// TwinCAT 3 PLC project Gantry
// ProgramVersion: 3.1.4023.0
// libraries:
//   Tc2_MC2, * (Beckhoff Automation GmbH)
//   Tc2_Standard, * (Beckhoff Automation GmbH)
//   Tc2_System, * (Beckhoff Automation GmbH)
//   Tc3_Module, * (Beckhoff Automation GmbH)
// project tree:
//   DUTs/ ST_PalletRecord.TcDUT
//   GVLs/ GVL_IO.TcGVL
//   / PlcTask.TcTTO
//   POUs/Devices/Actuator/ E_ActuatorCommand.TcDUT, E_ActuatorState.TcDUT, FB_Actuator.TcPOU
//   POUs/Devices/Axis/ E_AxisCommand.TcDUT, E_AxisState.TcDUT, FB_Axis.TcPOU
//   POUs/Devices/RFID/ E_RFIDCommand.TcDUT, E_RFIDState.TcDUT, FB_RFID.TcPOU
//   POUs/Interfaces/ I_GantryPallet.TcIO, I_GantryPart.TcIO
//   POUs/Modules/Gantry/ E_GantryCommand.TcDUT, E_GantryState.TcDUT, FB_Gantry.TcPOU
//   POUs/Modules/PalletStation/ E_PalletStationCommand.TcDUT, E_PalletStationState.TcDUT, FB_PalletStation.TcPOU
//   POUs/Modules/PartStation/ E_PartStationCommand.TcDUT, E_PartStationState.TcDUT, FB_PartStation.TcPOU
//   Program/ MAIN.TcPOU
// real-time tasks:
//   TASK PlcTask: cycle T#10ms, priority 20, ADS port 350
// motion (NC):
//   TASK NC-Task 1 SAF: cycle T#2ms, priority 4, ADS port 501
//   TASK NC-Task 1 SVB: cycle T#10ms, priority 8, ADS port 511
//   AXIS Gantry1X (id 1)
//     OtherSettings: AllowMotionCmdToSlave=true
//     encoder EncType=1
//     drive DrvType=5
//       Analog: TorqueSetpointScale=10, ScaleFactorActTorque=0.1
//       TimeComp: TaskDelayCycles=1
//     controller CtrType=1
//       CtrPara: PriorControlFactor=1
//         Observer: BandWidth=20
//   AXIS Gantry1Z (id 2)
//     OtherSettings: AllowMotionCmdToSlave=true
//     encoder EncType=1
//     drive DrvType=5
//       Analog: TorqueSetpointScale=10, ScaleFactorActTorque=0.1
//       TimeComp: TaskDelayCycles=1
//     controller CtrType=1
//       CtrPara: PriorControlFactor=1
//         Observer: BandWidth=20
//   AXIS Gantry2X (id 3)
//     OtherSettings: AllowMotionCmdToSlave=true
//     encoder EncType=1
//     drive DrvType=5
//       Analog: TorqueSetpointScale=10, ScaleFactorActTorque=0.1
//       TimeComp: TaskDelayCycles=1
//     controller CtrType=1
//       CtrPara: PriorControlFactor=1
//         Observer: BandWidth=20
//   AXIS Gantry2Z (id 4)
//     OtherSettings: AllowMotionCmdToSlave=true
//     encoder EncType=1
//     drive DrvType=5
//       Analog: TorqueSetpointScale=10, ScaleFactorActTorque=0.1
//       TimeComp: TaskDelayCycles=1
//     controller CtrType=1
//       CtrPara: PriorControlFactor=1
//         Observer: BandWidth=20
//   AXIS PalletConveyor (id 5)
//     OtherSettings: AllowMotionCmdToSlave=true
//     encoder EncType=1
//     drive DrvType=5
//       Analog: TorqueSetpointScale=10, ScaleFactorActTorque=0.1
//       TimeComp: TaskDelayCycles=1
//     controller CtrType=1
//       CtrPara: PriorControlFactor=1
//         Observer: BandWidth=20
//   AXIS PartConveyor1 (id 6)
//     OtherSettings: AllowMotionCmdToSlave=true
//     encoder EncType=1
//     drive DrvType=5
//       Analog: TorqueSetpointScale=10, ScaleFactorActTorque=0.1
//       TimeComp: TaskDelayCycles=1
//     controller CtrType=1
//       CtrPara: PriorControlFactor=1
//         Observer: BandWidth=20
//   AXIS PartConveyor2 (id 7)
//     OtherSettings: AllowMotionCmdToSlave=true
//     encoder EncType=1
//     drive DrvType=5
//       Analog: TorqueSetpointScale=10, ScaleFactorActTorque=0.1
//       TimeComp: TaskDelayCycles=1
//     controller CtrType=1
//       CtrPara: PriorControlFactor=1
//         Observer: BandWidth=20
// variable links:
//   Gantry/Gantry Instance <-> NC-Task 1 SAF/Axes/Gantry1X
//     PlcTask Inputs/GVL_IO.Gantry1X.NcToPlc <-> Outputs/ToPlc
//     PlcTask Outputs/GVL_IO.Gantry1X.PlcToNc <-> Inputs/FromPlc
//   Gantry/Gantry Instance <-> NC-Task 1 SAF/Axes/Gantry1Z
//     PlcTask Inputs/GVL_IO.Gantry1Z.NcToPlc <-> Outputs/ToPlc
//     PlcTask Outputs/GVL_IO.Gantry1Z.PlcToNc <-> Inputs/FromPlc
//   Gantry/Gantry Instance <-> NC-Task 1 SAF/Axes/Gantry2X
//     PlcTask Inputs/GVL_IO.Gantry2X.NcToPlc <-> Outputs/ToPlc
//     PlcTask Outputs/GVL_IO.Gantry2X.PlcToNc <-> Inputs/FromPlc
//   Gantry/Gantry Instance <-> NC-Task 1 SAF/Axes/Gantry2Z
//     PlcTask Inputs/GVL_IO.Gantry2Z.NcToPlc <-> Outputs/ToPlc
//     PlcTask Outputs/GVL_IO.Gantry2Z.PlcToNc <-> Inputs/FromPlc
//   Gantry/Gantry Instance <-> NC-Task 1 SAF/Axes/PalletConveyor
//     PlcTask Inputs/GVL_IO.PalletConveyor.NcToPlc <-> Outputs/ToPlc
//     PlcTask Outputs/GVL_IO.PalletConveyor.PlcToNc <-> Inputs/FromPlc
//   Gantry/Gantry Instance <-> NC-Task 1 SAF/Axes/PartConveyor1
//     PlcTask Inputs/GVL_IO.PartConveyor1.NcToPlc <-> Outputs/ToPlc
//     PlcTask Outputs/GVL_IO.PartConveyor1.PlcToNc <-> Inputs/FromPlc
//   Gantry/Gantry Instance <-> NC-Task 1 SAF/Axes/PartConveyor2
//     PlcTask Inputs/GVL_IO.PartConveyor2.NcToPlc <-> Outputs/ToPlc
//     PlcTask Outputs/GVL_IO.PartConveyor2.PlcToNc <-> Inputs/FromPlc

CONFIGURATION Gantry
    RESOURCE PLC ON TwinCAT3
        TASK PlcTask(INTERVAL := T#10ms, PRIORITY := 20);
        PROGRAM MAIN WITH PlcTask : MAIN;
    END_RESOURCE
END_CONFIGURATION

// ---- DUTs/ST_PalletRecord.TcDUT
TYPE ST_PalletRecord :
STRUCT
	ID				: STRING;
	Data			: ARRAY[1..100] OF STRING;
END_STRUCT
END_TYPE

// ---- POUs/Devices/Actuator/E_ActuatorCommand.TcDUT
{attribute 'qualified_only'}
{attribute 'strict'}
TYPE E_ActuatorCommand :
(
	None 		:= 0,
	Home		:= 1,
	Work		:= 2
) DINT;
END_TYPE

// ---- POUs/Devices/Actuator/E_ActuatorState.TcDUT
{attribute 'qualified_only'}
{attribute 'strict'}
TYPE E_ActuatorState :
(
	AtHome		:= 0, //Actuator at home
	AtWork		:= 1, //Actuator at work
	GoingToHome	:= 2, //Actuator going to home
	GoingToWork	:= 3 //Actuator going to work
) DINT;
END_TYPE

// ---- POUs/Devices/Axis/E_AxisCommand.TcDUT
{attribute 'qualified_only'}
{attribute 'strict'}
TYPE E_AxisCommand :
(
	None 				:= 0,
	TurnOn				:= 1,
	TurnOff				:= 2,
	ExecuteMoveAbs		:= 3,
	ExecuteMoveVel		:= 4,
	Stop				:= 5
) DINT;
END_TYPE

// ---- POUs/Devices/Axis/E_AxisState.TcDUT
{attribute 'qualified_only'}
{attribute 'strict'}
TYPE E_AxisState :
(
	Off					:= 0, //Axis is off
	Ready				:= 1, //Axis is ready/on
	Moving				:= 2, //Axis is moving to commanded position
	Stopping			:= 3, //Axis is stopping
	Stopped				:= 4, //Axis is stopped
	TurningOn			:= 5, //Axis is turning on
	TurningOff			:= 6 //Axis is turning off
) DINT;
END_TYPE

// ---- POUs/Devices/RFID/E_RFIDCommand.TcDUT
{attribute 'qualified_only'}
{attribute 'strict'}
TYPE E_RFIDCommand :
(
	None 		:= 0,
	Clear		:= 1,
	Read		:= 2
) DINT;
END_TYPE

// ---- POUs/Devices/RFID/E_RFIDState.TcDUT
{attribute 'qualified_only'}
{attribute 'strict'}
TYPE E_RFIDState :
(
	Idle			:= 0,
	Clearing		:= 1,
	Reading			:= 2,
	Completing		:= 3
);
END_TYPE

// ---- POUs/Modules/Gantry/E_GantryCommand.TcDUT
{attribute 'qualified_only'}
{attribute 'strict'}
TYPE E_GantryCommand :
(
	None 			:= 0,
	TurnOn			:= 1,
	TurnOff			:= 2,
	Pick			:= 3,
	Place			:= 4,
	Home			:= 5,
	Abort			:= 6
) DINT;
END_TYPE

// ---- POUs/Modules/Gantry/E_GantryState.TcDUT
{attribute 'qualified_only'}
{attribute 'strict'}
TYPE E_GantryState :
(
	Idle 			:= 0,
	TurningOn		:= 1,
	TurningOff		:= 2,
	Ready			:= 3,
	Picking			:= 4,
	Placing			:= 5,
	Homing			:= 6,
	Aborting		:= 7
) DINT;
END_TYPE

// ---- POUs/Modules/PalletStation/E_PalletStationCommand.TcDUT
{attribute 'qualified_only'}
{attribute 'strict'}
TYPE E_PalletStationCommand :
(
	None 			:= 0,
	Start			:= 1,
	Stop			:= 2,
	Home			:= 3,
	Abort			:= 4
) DINT;
END_TYPE

// ---- POUs/Modules/PalletStation/E_PalletStationState.TcDUT
{attribute 'qualified_only'}
{attribute 'strict'}
TYPE E_PalletStationState :
(
	Idle 			:= 0,
	Starting		:= 1,
	Running			:= 2,
	Stopping		:= 3,
	Homing			:= 4,
	Aborting		:= 5
);
END_TYPE

// ---- POUs/Modules/PartStation/E_PartStationCommand.TcDUT
{attribute 'qualified_only'}
{attribute 'strict'}
TYPE E_PartStationCommand :
(
	None 			:= 0,
	Start			:= 1,
	Stop			:= 2,
	Abort			:= 3
) DINT;
END_TYPE

// ---- POUs/Modules/PartStation/E_PartStationState.TcDUT
{attribute 'qualified_only'}
{attribute 'strict'}
TYPE E_PartStationState :
(
	Idle 			:= 0,
	Starting		:= 1,
	Running			:= 2,
	Stopping		:= 3,
	Stopped			:= 4,
	Aborting		:= 5
);
END_TYPE

// ---- GVLs/GVL_IO.TcGVL
{attribute 'qualified_only'}
VAR_GLOBAL
	Gantry1X			: AXIS_REF;
	Gantry1Z			: AXIS_REF;
	Gantry2X			: AXIS_REF;
	Gantry2Z			: AXIS_REF;
	PalletConveyor		: AXIS_REF;
	PartConveyor1		: AXIS_REF;
	PartConveyor2		: AXIS_REF;
	
	PalletRecord		: ARRAY[0..100] OF ST_PalletRecord;
	ActiveRecord		: DINT;
END_VAR

// ---- POUs/Interfaces/I_GantryPallet.TcIO
INTERFACE I_GantryPallet

PROPERTY PalletReady : BOOL
GET
END_GET
END_PROPERTY

END_INTERFACE

// ---- POUs/Interfaces/I_GantryPart.TcIO
INTERFACE I_GantryPart

PROPERTY PartPicked : BOOL
GET
END_GET
END_PROPERTY

PROPERTY PartReady : BOOL
GET
END_GET
END_PROPERTY

END_INTERFACE

// ---- Program/MAIN.TcPOU
PROGRAM MAIN
VAR
	inpSim					: BOOL := TRUE;
	
	PalletStation			: FB_PalletStation;
	Part1Station			: FB_PartStation;
	Part2Station			: FB_PartStation;
	Gantry1					: FB_Gantry;
	Gantry2					: FB_Gantry;
	
	Gantry1NextPlace		: DINT;
	Gantry2NextPlace		: DINT;
	
	Start					: BOOL;
	Abort					: BOOL;
	Home					: BOOL;
END_VAR

IF inpSim THEN
	Simulate();
END_IF

PalletStation(Axis := GVL_IO.PalletConveyor, 
		inpPalletRecord := GVL_IO.PalletRecord,
		inpActiveRecord := GVL_IO.ActiveRecord,
		ipGantry1 := Gantry1, 
		ipGantry2 := Gantry2);
Part1Station(Axis := GVL_IO.PartConveyor1, 
		ipGantry := Gantry1);
Part2Station(Axis := GVL_IO.PartConveyor2, 
		ipGantry := Gantry2);

Gantry1(AxisX := GVL_IO.Gantry1X,
		AxisZ := GVL_IO.Gantry1Z,
		ipPart := Part1Station,
		ipPallet := PalletStation,
		inpPalletRecord := GVL_IO.PalletRecord,
		inpActiveRecord := GVL_IO.ActiveRecord,
		inpDataIndex1 := 1,
		inpDataIndex2 := 2,
		inpDataIndex3 := 3,
		inpDataIndex4 := 4,
		inpDataIndex5 := 5,
		inpDataIndex6 := 6,
		inpX_HomePos := 0,		
		inpX_PickPos := 100,	
		inpX_PlacePos1 := 2050,
		inpX_PlacePos2 := 2100,
		inpX_PlacePos3 := 2150,
		inpX_PrePlacePos := 2000,
		inpZ_HomePos := 0,
		inpZ_PickPos := 3500,
		inpZ_PlacePos := 3000,
		inpZ_PrePickPos := 2500); //Positions are hardcoded to make simulation easier. Best practice would be to use an array with recipe management.

Gantry2(AxisX := GVL_IO.Gantry2X,
		AxisZ := GVL_IO.Gantry2Z,
		ipPart := Part2Station,
		ipPallet := PalletStation,
		inpPalletRecord := GVL_IO.PalletRecord,
		inpActiveRecord := GVL_IO.ActiveRecord,
		inpDataIndex1 := 12,
		inpDataIndex2 := 11,
		inpDataIndex3 := 10,
		inpDataIndex4 := 9,
		inpDataIndex5 := 8,
		inpDataIndex6 := 7,
		inpX_HomePos := 0,		
		inpX_PickPos := 100,	
		inpX_PlacePos1 := 2700,
		inpX_PlacePos2 := 2750,
		inpX_PlacePos3 := 2800,
		inpX_PrePlacePos := 1900,
		inpZ_HomePos := 0,
		inpZ_PickPos := 3500,
		inpZ_PlacePos := 3000,
		inpZ_PrePickPos := 2500); //Positions are hardcoded to make simulation easier. Best practice would be to use an array with recipe management.

//Start all modules		
IF Start THEN
	PalletStation.cmd := E_PalletStationCommand.Start;
	Part1Station.cmd := E_PartStationCommand.Start;
	Part2Station.cmd := E_PartStationCommand.Start;
	Gantry1.cmd := E_GantryCommand.TurnOn;
	Gantry2.cmd := E_GantryCommand.TurnOn;
	Start := FALSE;
END_IF

//Abort all modules
IF Abort THEN
	PalletStation.cmd := E_PalletStationCommand.Abort;
	Part1Station.cmd := E_PartStationCommand.Abort;
	Part2Station.cmd := E_PartStationCommand.Abort;
	Gantry1.cmd := E_GantryCommand.Abort;
	Gantry2.cmd := E_GantryCommand.Abort;
	Abort := FALSE;
END_IF

//Home all modules
IF Home THEN
	IF (PalletStation.stsState = E_PalletStationState.Idle AND 
		Gantry1.stsState = E_GantryState.Idle AND 
		Gantry2.stsState = E_GantryState.Idle) 
	THEN
		PalletStation.cmd := E_PalletStationCommand.Home;
		Gantry1.cmd := E_GantryCommand.Home;
		Gantry2.cmd := E_GantryCommand.Home;
		Home := FALSE;
	END_IF
END_IF

METHOD Simulate : BOOL
VAR_INPUT
END_VAR
GVL_IO.PalletRecord[5].ID := '12345';
END_METHOD

END_PROGRAM

// ---- POUs/Modules/PalletStation/FB_PalletStation.TcPOU
FUNCTION_BLOCK FB_PalletStation IMPLEMENTS I_GantryPallet
VAR_INPUT
	Axis				: REFERENCE TO AXIS_REF;
	ipGantry1			: I_GantryPallet;
	ipGantry2			: I_GantryPallet;
	cmd					: E_PalletStationCommand := E_PalletStationCommand.None;
	
	inpPalletRecord		: REFERENCE TO ARRAY[0..100] OF ST_PalletRecord;
	inpActiveRecord		: REFERENCE TO DINT;	
	inpSim				: BOOL := TRUE;
	inpPalletPresent	AT %I* : BOOL;
END_VAR
VAR_OUTPUT
	stsState			: E_PalletStationState := E_PalletStationState.Idle;
	stsCurrentStep		: DINT;
END_VAR
VAR
	//Devices
	Conveyor			: FB_Axis;
	PalletStop			: FB_Actuator;
	RFID				: FB_RFID;
	
	DepartureTimer		: TON;
	DepartureDelayTime	: TIME := T#3S;
	PP_DepartSimTimer	: TON;
	PP_ArriveSimTimer	: TON;
	
	rtStarting			: R_TRIG;
	rtStopping			: R_TRIG;
	rtHoming			: R_TRIG;
	rtPalletPresent		: R_TRIG;

	i					: DINT;	
	j					: DINT;
	Gantry1Clear		: BOOL;
	Gantry2Clear		: BOOL;
END_VAR
VAR CONSTANT
	NULL_RECORD			: ARRAY[1..100] OF STRING;
END_VAR

Map();
Status();
StateMachine();

METHOD Aborting : BOOL
VAR_INPUT
END_VAR
Conveyor.cmd := E_AxisCommand.Stop;
stsCurrentStep := 0;
END_METHOD

METHOD Homing : BOOL
VAR_INPUT
END_VAR
CASE stsCurrentStep OF
	4000: //Clear RFID and active record
		RFID.cmd := E_RFIDCommand.Clear;
		inpActiveRecord := 0;
		IF RFID.stsCurrentID = '' THEN
			stsCurrentStep := 4010;
		END_IF
	4010: //Extend pallet stop
		PalletStop.cmd := E_ActuatorCommand.Work;
		IF PalletStop.stsState = E_ActuatorState.AtWork THEN
			stsCurrentStep := 4020;
		END_IF
	4020: //Stop conveyor
		Conveyor.cmd := E_AxisCommand.Stop;
		IF Conveyor.stsVelocity = 0 THEN
			stsCurrentStep := 0;
		END_IF
END_CASE
END_METHOD

METHOD Map : BOOL
VAR_INPUT
END_VAR
Conveyor(Axis := Axis);
PalletStop();
RFID();

DepartureTimer(IN := stsCurrentStep = 3050 AND NOT inpPalletPresent, PT := DepartureDelayTime);

Gantry1Clear := ipGantry1.PalletReady;
Gantry2Clear := ipGantry2.PalletReady;
END_METHOD

{warning 'add property implementation'}
PROPERTY PalletReady : BOOL
GET
PalletReady := inpPalletPresent AND Gantry1Clear AND Gantry2Clear AND PalletStop.stsState = E_ActuatorState.AtWork;
END_GET
END_PROPERTY

METHOD Running : BOOL
VAR_INPUT
END_VAR
CASE stsCurrentStep OF
	3000: //Read RFID
		RFID.cmd := E_RFIDCommand.Read;
		IF RFID.stsCurrentID <> '' THEN
			stsCurrentStep := 3010;
		END_IF
	3010: //Clear associated data
		FOR i := 1 TO 100 DO
			IF inpPalletRecord[i].ID = RFID.stsCurrentID THEN
				inpPalletRecord[i].Data := NULL_RECORD;
				inpActiveRecord := i;
				stsCurrentStep := 3020;
			END_IF
		END_FOR
	3020: //Wait for all 12 records to populate
		IF (inpPalletRecord[inpActiveRecord].Data[1] <> '' AND
			inpPalletRecord[inpActiveRecord].Data[2] <> '' AND
			inpPalletRecord[inpActiveRecord].Data[3] <> '' AND
			inpPalletRecord[inpActiveRecord].Data[4] <> '' AND
			inpPalletRecord[inpActiveRecord].Data[5] <> '' AND
			inpPalletRecord[inpActiveRecord].Data[6] <> '' AND
			inpPalletRecord[inpActiveRecord].Data[7] <> '' AND
			inpPalletRecord[inpActiveRecord].Data[8] <> '' AND
			inpPalletRecord[inpActiveRecord].Data[9] <> '' AND
			inpPalletRecord[inpActiveRecord].Data[10] <> '' AND
			inpPalletRecord[inpActiveRecord].Data[11] <> '' AND
			inpPalletRecord[inpActiveRecord].Data[12] <> '')
		THEN
			inpActiveRecord := 0;
			stsCurrentStep := 3030;
		END_IF
	3030: //Wait for gantries to clear station
		IF Gantry1Clear AND Gantry2Clear THEN
			stsCurrentStep := 3040;
		END_IF
	3040: //Release pallet
		PalletStop.cmd := E_ActuatorCommand.Home;
		IF PalletStop.stsState = E_ActuatorState.AtHome THEN
			stsCurrentStep := 3050;
		END_IF
	3050: //Wait for pallet to leave
		IF DepartureTimer.Q THEN
			stsCurrentStep := 3060;
		END_IF
	3060: //Extend pallet stop
		PalletStop.cmd := E_ActuatorCommand.Work;
		IF PalletStop.stsState = E_ActuatorState.AtWork THEN
			stsCurrentStep := 3070;
		END_IF
	3070: //Clear RFID
		RFID.cmd := E_RFIDCommand.Clear;
		IF RFID.stsCurrentID = '' THEN
			stsCurrentStep := 0;
		END_IF
END_CASE
END_METHOD

METHOD Simulate : BOOL
VAR_INPUT
END_VAR
PP_DepartSimTimer(IN := stsCurrentStep = 3050, PT := T#5S);
inpPalletPresent R= PP_DepartSimTimer.Q;

PP_ArriveSimTimer(IN := stsState = E_PalletStationState.Running AND NOT inpPalletPresent, PT := T#10S);
inpPalletPresent S= PP_ArriveSimTimer.Q;
END_METHOD

METHOD Starting : BOOL
VAR_INPUT
END_VAR
CASE stsCurrentStep OF
	1000: //Clear RFID
		RFID.cmd := E_RFIDCommand.Clear;
		IF RFID.stsCurrentID = '' THEN
			stsCurrentStep := 1010;
		END_IF
	1010: //Extend pallet stop
		PalletStop.cmd := E_ActuatorCommand.Work;
		IF PalletStop.stsState = E_ActuatorState.AtWork THEN
			stsCurrentStep := 1020;
		END_IF
	1020: //Turn on conveyor
		Conveyor.cmd := E_AxisCommand.TurnOn;
		IF Conveyor.stsState = E_AxisState.Ready THEN
			stsCurrentStep := 1030;
		END_IF
	1030: //Run conveyor at 100 mm/s (arbitrary value for project)
		Conveyor.inpVelocity := 100;
		Conveyor.cmd := E_AxisCommand.ExecuteMoveVel;
		IF Conveyor.stsVelocity > 0 THEN
			stsCurrentStep := 0;
		END_IF
END_CASE
END_METHOD

METHOD StateMachine : BOOL
VAR_INPUT
END_VAR
IF inpSim THEN
	Simulate();
END_IF

CASE stsState OF
	E_PalletStationState.Idle: //Station idle and ready for command
		IF cmd = E_PalletStationCommand.Start THEN
			stsState := E_PalletStationState.Starting;
		ELSIF cmd = E_PalletStationCommand.Home THEN
			stsState := E_PalletStationState.Homing;
		END_IF
	E_PalletStationState.Homing: //Return station to home state
		Homing();
		IF stsCurrentStep = 0 AND PalletStop.stsState = E_ActuatorState.AtWork THEN
			stsState := E_PalletStationState.Idle;
		END_IF
	E_PalletStationState.Starting: //Start conveyor and ready to process
		Starting();
		IF stsCurrentStep = 0 AND Conveyor.stsVelocity > 0 AND PalletStop.stsState = E_ActuatorState.AtWork THEN
			stsState := E_PalletStationState.Running;
		END_IF
	E_PalletStationState.Running: //Station is running and ready to receive pallet
		Running();
		IF cmd = E_PalletStationCommand.Stop THEN
			Stopping();
			stsState := E_PalletStationState.Stopping;
		END_IF
	E_PalletStationState.Stopping: //Station is stopping
		Stopping();
		IF stsCurrentStep = 0 AND Conveyor.stsVelocity = 0 AND PalletStop.stsState = E_ActuatorState.AtWork THEN
			stsState := E_PalletStationState.Idle;
		END_IF
	E_PalletStationState.Aborting: //Abort all station activity
		Aborting();
		IF stsCurrentStep = 0 AND Conveyor.stsVelocity = 0 THEN
			stsState := E_PalletStationState.Idle;
		END_IF		
END_CASE

IF cmd = E_PalletStationCommand.Abort THEN
	stsState := E_PalletStationState.Aborting;
END_IF

cmd := E_PalletStationCommand.None;
END_METHOD

METHOD Status : BOOL
VAR_INPUT
END_VAR
//State transition one shots
rtStarting(CLK := stsState = E_PalletStationState.Starting);
IF rtStarting.Q THEN
	stsCurrentStep := 1000;
END_IF

rtStopping(CLK := stsState = E_PalletStationState.Stopping);
IF rtStopping.Q THEN
	stsCurrentStep := 2000;
END_IF

rtHoming(CLK := stsState = E_PalletStationState.Homing);
IF rtHoming.Q THEN
	stsCurrentStep := 4000;
END_IF

rtPalletPresent(CLK := inpPalletPresent AND stsState <> E_PalletStationState.Homing AND stsCurrentStep = 0);
IF rtPalletPresent.Q THEN
	stsCurrentStep := 3000;
END_IF
END_METHOD

METHOD Stopping : BOOL
VAR_INPUT
END_VAR

VAR
	END_IFCASE: INT;
END_VAR
CASE stsCurrentStep OF
	2000: //Clear RFID
		RFID.cmd := E_RFIDCommand.Clear;
		IF RFID.stsCurrentID = '' THEN
			stsCurrentStep := 2010;
		END_IF
	2010: //Extend pallet stop
		PalletStop.cmd := E_ActuatorCommand.Work;
		IF PalletStop.stsState = E_ActuatorState.AtWork THEN
			stsCurrentStep := 2020;
		END_IF
	2020: //Stop conveyor
		Conveyor.cmd := E_AxisCommand.Stop;
		IF Conveyor.stsVelocity = 0 THEN
			stsCurrentStep := 0;
		END_IF
END_CASE
END_METHOD

END_FUNCTION_BLOCK

// ---- POUs/Devices/Axis/FB_Axis.TcPOU
FUNCTION_BLOCK FB_Axis
VAR_INPUT
	Axis				: REFERENCE TO AXIS_REF;
	cmd					: E_AxisCommand := E_AxisCommand.None;
	
	inpSim				: BOOL := TRUE;
	inpPosition			: LREAL;
	inpVelocity			: LREAL := 500.0;
	inpAcceleration		: LREAL := 100.0;
	inpDeceleration		: LREAL := 100.0;
END_VAR
VAR_OUTPUT
	stsState			: E_AxisState := E_AxisState.Off;
	stsFaultCode		: DINT;
	stsPowerOn			: BOOL;
	stsPosition			: LREAL;
	stsVelocity			: LREAL;
END_VAR
VAR
	PowerOn				: MC_Power;
	MoveAbs				: MC_MoveAbsolute;
	MoveVel				: MC_MoveVelocity;
	MoveStop			: MC_Stop;

	PowerOnTimer		: TON;
	StartTimer			: TON;
	StopTimer			: TON;
	PowerOnSimTime		: TIME := T#3S;
	StartSimTime		: TIME := T#3S;
	StopSimTime			: TIME := T#3S;
	PowerOnFailTime		: TIME := T#5S;
	StartFailTime		: TIME := T#5S;
	StopFailTime		: TIME := T#5S;
END_VAR

Map();
Status();
StateMachine();
Control();

METHOD Control : BOOL
VAR_INPUT
END_VAR
IF stsState = E_AxisState.TurningOn THEN
	PowerOn.Enable := TRUE;
	PowerOn.Enable_Negative := TRUE;
	PowerOn.Enable_Positive := TRUE;
END_IF

IF stsState = E_AxisState.TurningOff THEN
	PowerOn.Enable := FALSE;
	PowerOn.Enable_Negative := FALSE;
	PowerOn.Enable_Positive := FALSE;
END_IF

IF stsState = E_AxisState.Stopping THEN
	MoveStop.Execute := TRUE;
END_IF
END_METHOD

METHOD Map : BOOL
VAR_INPUT
END_VAR
MoveAbs(Axis := Axis, Position := inpPosition, Velocity := inpVelocity, Acceleration := inpAcceleration, Deceleration := inpDeceleration);
MoveVel(Axis := Axis, Velocity := inpVelocity, Acceleration := inpAcceleration, Deceleration := inpDeceleration);
MoveStop(Axis := Axis);
PowerOn(Axis := Axis);
END_METHOD

METHOD StateMachine : BOOL
VAR_INPUT
END_VAR
CASE stsState OF
	E_AxisState.Off:
		IF cmd = E_AxisCommand.TurnOn THEN
			stsState := E_AxisState.TurningOn;
		END_IF
	E_AxisState.TurningOn:
		IF stsPowerOn THEN
			stsState := E_AxisState.Ready;
		END_IF
	E_AxisState.Ready:
		IF cmd = E_AxisCommand.ExecuteMoveAbs THEN
			MoveAbs.Execute := TRUE;
		ELSIF cmd = E_AxisCommand.ExecuteMoveVel THEN
			MoveVel.Execute := TRUE;
		ELSIF cmd = E_AxisCommand.Stop THEN
			MoveAbs.Execute := FALSE;
			MoveVel.Execute := FALSE;
			stsState := E_AxisState.Stopping;
		END_IF
		IF MoveAbs.Busy THEN
			MoveAbs.Execute := FALSE;
			MoveVel.Execute := FALSE;
			stsState := E_AxisState.Moving;
		END_IF
	E_AxisState.Moving:
		IF MoveAbs.Done THEN
			stsState := E_AxisState.Ready;
		ELSIF cmd = E_AxisCommand.Stop THEN
			stsState := E_AxisState.Stopping;
		END_IF
	E_AxisState.Stopping:
		IF NOT MoveAbs.Busy THEN
			MoveStop.Execute := FALSE;
			stsState := E_AxisState.Ready;
		END_IF
	E_AxisState.TurningOff:
		IF NOT stsPowerOn THEN
			stsState := E_AxisState.Off;
		END_IF
END_CASE

IF cmd = E_AxisCommand.TurnOff THEN
	stsState := E_AxisState.TurningOff;
END_IF

cmd := E_AxisCommand.None;
END_METHOD

METHOD Status : BOOL
VAR_INPUT
END_VAR
stsPowerOn := PowerOn.Status;
stsPosition := Axis.NcToPlc.ActPos;
stsVelocity := Axis.NcToPlc.ActVelo;
END_METHOD

END_FUNCTION_BLOCK

// ---- POUs/Devices/Actuator/FB_Actuator.TcPOU
FUNCTION_BLOCK FB_Actuator
VAR_INPUT
	cmd					: E_ActuatorCommand := E_ActuatorCommand.None;
	
	inpSim				: BOOL := TRUE;
	inpHome				AT %I* : BOOL;
	inpWork				AT %I* : BOOL;
END_VAR
VAR_OUTPUT
	stsState			: E_ActuatorState := E_ActuatorState.AtHome;
	stsFaultCode		: DINT;
	
	outHome				AT %Q* : BOOL;
	outWork				AT %Q* : BOOL;
END_VAR
VAR
	WorkTimer			: TON;
	HomeTimer			: TON;
	WorkSimTime			: TIME := T#2S;
	HomeSimTime			: TIME := T#2S;
	WorkFailTime		: TIME := T#10S;
	HomeFailTime		: TIME := T#10S;
END_VAR

Faults();
StateMachine();
Control();

METHOD Control : BOOL
VAR_INPUT
END_VAR
outHome := stsState = (E_ActuatorState.AtHome OR E_ActuatorState.GoingToHome);
outWork := stsState = (E_ActuatorState.AtWork OR E_ActuatorState.GoingToWork);
END_METHOD

METHOD Faults : BOOL
VAR_INPUT
END_VAR
WorkTimer(IN := stsState = E_ActuatorState.GoingToWork, PT := WorkFailTime);
HomeTimer(IN := stsState = E_ActuatorState.GoingToHome, PT := HomeFailTime);
IF WorkTimer.Q THEN
	stsFaultCode := 100;
ELSIF HomeTImer.Q THEN
	stsFaultCode := 200;
ELSE
	stsFaultCode := 0;
END_IF
END_METHOD

METHOD Simulate : BOOL
VAR_INPUT
END_VAR
inpWork := outWork AND WorkTimer.ET >= WorkSimTime;
inpHome := outHome AND HomeTimer.ET >= HomeSimTime;
END_METHOD

METHOD StateMachine : BOOL
VAR_INPUT
END_VAR
IF inpSim THEN
	Simulate();
END_IF

CASE stsState OF
	E_ActuatorState.AtHome:
		IF cmd = E_ActuatorCommand.Work THEN
			stsState := E_ActuatorState.GoingToWork;
		END_IF
	E_ActuatorState.AtWork:
		IF cmd = E_ActuatorCommand.Home THEN
			stsState := E_ActuatorState.GoingToHome;
		END_IF
	E_ActuatorState.GoingToHome:
		IF inpHome THEN
			stsState := E_ActuatorState.AtHome;
		ELSIF cmd = E_ActuatorCommand.Work THEN
			stsState := E_ActuatorState.GoingToWork;
		END_IF
	E_ActuatorState.GoingToWork:
		IF inpWork THEN
			stsState := E_ActuatorState.AtWork;
		ELSIF cmd = E_ActuatorCommand.Home THEN
			stsState := E_ActuatorState.GoingToHome;
		END_IF
END_CASE
END_METHOD

END_FUNCTION_BLOCK

// ---- POUs/Devices/RFID/FB_RFID.TcPOU
FUNCTION_BLOCK FB_RFID
VAR_INPUT
	cmd					: E_RFIDCommand := E_RFIDCommand.None;
	cmdReset			: BOOL;
	inpSimID			: STRING := '12345';
	
	inpSim				: BOOL := TRUE;
	inpID				AT %I* : STRING;
END_VAR
VAR_OUTPUT
	stsState			: E_RFIDState := E_RFIDState.Idle;
	stsFaultCode		: DINT;
	stsCurrentID		: STRING;
	
	outScan				AT %Q* : BOOL;
	outResetScanner		AT %Q* : BOOL;
END_VAR
VAR
	ReadTimer			: TON;
	ReadSimTime			: TIME := T#5S;
	ReadFailTime		: TIME := T#30S;
END_VAR
VAR CONSTANT
	NULL_ID				: STRING := '';
END_VAR

Faults();
StateMachine();
Control();

METHOD Control : BOOL
VAR_INPUT
END_VAR
outScan := stsState = E_RFIDState.Reading;
outResetScanner := stsState = E_RFIDState.Completing;
END_METHOD

METHOD Faults : BOOL
VAR_INPUT
END_VAR
ReadTimer(IN := stsState = E_RFIDState.Reading, PT := ReadFailTime);
IF ReadTimer.Q THEN
	stsFaultCode := 100;
ELSE
	stsFaultCode := 0;
END_IF
END_METHOD

METHOD Simulate : BOOL
VAR_INPUT
END_VAR
IF outScan AND ReadTimer.ET >= ReadSimTime THEN
	inpID := inpSimID;
END_IF

IF outResetScanner THEN
	inpID := NULL_ID;
END_IF
END_METHOD

METHOD StateMachine : BOOL
VAR_INPUT
END_VAR
IF inpSim THEN
	Simulate();
END_IF

CASE stsState OF
	E_RFIDState.Idle:
		IF cmd = E_RFIDCommand.Clear THEN
			stsState := E_RFIDState.Clearing;
		ELSIF cmd = E_RFIDCommand.Read THEN
			stsState := E_RFIDState.Reading;
		END_IF
	E_RFIDState.Clearing:
		stsCurrentID := NULL_ID;
		IF stsCurrentID = NULL_ID THEN
			stsState := E_RFIDState.Idle;
		END_IF
	E_RFIDState.Reading:
		IF inpID <> NULL_ID THEN
			stsCurrentID := inpID;
			stsState := E_RFIDState.Completing;
		ELSIF stsFaultCode <> 0 AND cmdReset THEN
			stsState := E_RFIDState.Idle;
		END_IF
	E_RFIDState.Completing:
		IF inpID = NULL_ID THEN
			stsState := E_RFIDState.Idle;
		END_IF
END_CASE

cmd := E_RFIDCommand.None;
cmdReset := FALSE;
END_METHOD

END_FUNCTION_BLOCK

// ---- POUs/Modules/PartStation/FB_PartStation.TcPOU
FUNCTION_BLOCK FB_PartStation IMPLEMENTS I_GantryPart
VAR_INPUT
	Axis				: REFERENCE TO AXIS_REF;
	ipGantry			: I_GantryPart;
	cmd					: E_PartStationCommand := E_PartStationCommand.None;
	
	inpSim				: BOOL := TRUE;
	inpPartPresent		AT %I* : BOOL;
END_VAR
VAR_OUTPUT
	stsState			: E_PartStationState := E_PartStationState.Idle;
	stsCurrentStep		: DINT;
END_VAR
VAR
	//Devices
	Conveyor			: FB_Axis;
	
	DebounceTimer		: TON;
	DebounceTime		: TIME := T#500MS;
	PP_DepartSimTimer	: TON;
	PP_ArriveSimTimer	: TON;
	
	rtStarting			: R_TRIG;
	rtStopping			: R_TRIG;
	rtPartPresent		: R_TRIG;

	GantryClear			: BOOL;
	GantryPickComplete	: BOOL;
END_VAR

Map();
Status();
StateMachine();

METHOD Aborting : BOOL
VAR_INPUT
END_VAR
Conveyor.cmd := E_AxisCommand.Stop;
stsCurrentStep := 0;
END_METHOD

METHOD Map : BOOL
VAR_INPUT
END_VAR
Conveyor(Axis := Axis);

DebounceTimer(IN := inpPartPresent, PT := DebounceTime);

GantryClear := ipGantry.PartReady;
GantryPickComplete := ipGantry.PartPicked;
END_METHOD

{warning 'add property implementation'}
PROPERTY PartPicked : BOOL
GET
PartPicked := NOT inpPartPresent;
END_GET
END_PROPERTY

{warning 'add property implementation'}
PROPERTY PartReady : BOOL
GET
PartReady := inpPartPresent AND Conveyor.stsVelocity = 0;
END_GET
END_PROPERTY

METHOD Simulate : BOOL
VAR_INPUT
END_VAR
rtPartPresent(CLK := GantryPickComplete);
inpPartPresent R= rtPartPresent.Q;

PP_ArriveSimTimer(IN := stsState = E_PartStationState.Running AND NOT inpPartPresent, PT := T#5S);
inpPartPresent S= PP_ArriveSimTimer.Q;
END_METHOD

METHOD Starting : BOOL
VAR_INPUT
END_VAR
CASE stsCurrentStep OF
	1000: //Turn on conveyor servo
		Conveyor.cmd := E_AxisCommand.TurnOn;
		IF Conveyor.stsState = E_AxisState.Ready THEN
			stsCurrentStep := 1010;
		END_IF
	1010: //Start conveyor at 100 mm/s (arbitrary value)
		Conveyor.inpVelocity := 100;
		Conveyor.cmd := E_AxisCommand.ExecuteMoveVel;
		IF Conveyor.stsVelocity > 0 THEN
			stsCurrentStep := 0;
		END_IF
END_CASE
END_METHOD

METHOD StateMachine : BOOL
VAR_INPUT
END_VAR
IF inpSim THEN
	Simulate();
END_IF

CASE stsState OF
	E_PartStationState.Idle: //Station is idle and ready for command
		IF cmd = E_PartStationCommand.Start THEN
			stsState := E_PartStationState.Starting;
		END_IF
	E_PartStationState.Starting: //Start conveyor and ready for parts
		Starting();
		IF stsCurrentStep = 0 AND Conveyor.stsVelocity > 0 THEN
			stsState := E_PartStationState.Running;
		END_IF
	E_PartStationState.Running: //Running and waiting for part present sensor
		IF DebounceTimer.Q THEN
			Stopping();
			stsState := E_PartStationState.Stopping;
		END_IF
	E_PartStationState.Stopping: //Stopping conveyor
		Stopping();
		IF stsCurrentStep = 0 AND Conveyor.stsVelocity = 0 THEN
			stsState := E_PartStationState.Stopped;
		END_IF
	E_PartStationState.Stopped: //Conveyor stopped. waiting for part pick
		IF NOT inpPartPresent AND GantryClear THEN
			Starting();
			stsState := E_PartStationState.Starting;
		END_IF
	E_PartStationState.Aborting: //Abort all station activity
		Aborting();
		IF stsCurrentStep = 0 AND Conveyor.stsVelocity = 0 THEN
			stsState := E_PartStationState.Idle;
		END_IF
END_CASE

IF cmd = E_PartStationCommand.Abort THEN
	stsState := E_PartStationState.Aborting;
END_IF

cmd := E_PartStationCommand.None;
END_METHOD

METHOD Status : BOOL
VAR_INPUT
END_VAR
//State transition one shots
rtStarting(CLK := stsState = E_PalletStationState.Starting);
IF rtStarting.Q THEN
	stsCurrentStep := 1000;
END_IF

rtStopping(CLK := stsState = E_PartStationState.Stopping);
IF rtStopping.Q THEN
	stsCurrentStep := 2000;
END_IF
END_METHOD

METHOD Stopping : BOOL
VAR_INPUT
END_VAR

VAR
	END_IFCASE: INT;
END_VAR
CASE stsCurrentStep OF
	2000: //Stop conveyor
		Conveyor.cmd := E_AxisCommand.Stop;
		IF Conveyor.stsVelocity = 0 THEN
			stsCurrentStep := 0;
		END_IF
END_CASE
END_METHOD

END_FUNCTION_BLOCK

// ---- POUs/Modules/Gantry/FB_Gantry.TcPOU
FUNCTION_BLOCK FB_Gantry IMPLEMENTS I_GantryPallet,I_GantryPart
VAR_INPUT
	AxisX				: REFERENCE TO AXIS_REF;
	AxisZ				: REFERENCE TO AXIS_REF;			
	ipPallet			: I_GantryPallet;
	ipPart				: I_GantryPart;
	
	cmd					: E_GantryCommand := E_GantryCommand.None;
	
	inpPalletRecord		: REFERENCE TO ARRAY[0..100] OF ST_PalletRecord;
	inpActiveRecord		: REFERENCE TO DINT;
	inpDataIndex1		: DINT;
	inpDataIndex2		: DINT;
	inpDataIndex3		: DINT;
	inpDataIndex4		: DINT;
	inpDataIndex5		: DINT;
	inpDataIndex6		: DINT;
	
	inpX_HomePos		: LREAL;
	inpX_PickPos		: LREAL;
	inpX_PlacePos1		: LREAL;
	inpX_PlacePos2		: LREAL;
	inpX_PlacePos3		: LREAL;
	inpX_PrePlacePos	: LREAL;
	inpZ_HomePos		: LREAL;
	inpZ_PickPos		: LREAL;
	inpZ_PlacePos		: LREAL;
	inpZ_PrePickPos		: LREAL;
END_VAR
VAR_OUTPUT
	stsState			: E_GantryState := E_GantryState.Idle;
	stsCurrentStep		: DINT;
END_VAR
VAR
	//Devices
	X_Axis				: FB_Axis;
	Z_Axis				: FB_Axis;
	Magnet				: FB_Actuator;
	Gripper				: FB_Actuator;
	
	rtTurningOn			: R_TRIG;
	rtTurningOff		: R_TRIG;
	rtPicking			: R_TRIG;
	rtPlacing			: R_TRIG;
	rtHoming			: R_TRIG;
	rtPartPresent		: R_TRIG;

	PalletConvReady		: BOOL;
	PartConvReady		: BOOL;
	
	NextPlaceIndex		: DINT;
	DataIndex1			: DINT;
	DataIndex2			: DINT;
END_VAR

Map();
Status();
StateMachine();

METHOD Aborting : BOOL
VAR_INPUT
END_VAR
X_Axis.cmd := E_AxisCommand.Stop;
Z_Axis.cmd := E_AxisCommand.Stop;
stsCurrentStep := 0;
END_METHOD

METHOD Homing : BOOL
VAR_INPUT
END_VAR
CASE stsCurrentStep OF
	5000: //Gripper and magnets to home position
		Magnet.cmd := E_ActuatorCommand.Home;
		Gripper.cmd := E_ActuatorCommand.Home;
		IF Magnet.stsState = E_ActuatorState.AtHome AND Gripper.stsState = E_ActuatorState.AtHome THEN
			stsCurrentStep := 5010;
		END_IF
	5010: //Turn on axes
		X_Axis.cmd := E_AxisCommand.TurnOn;
		Z_Axis.cmd := E_AxisCommand.TurnOn;
		IF X_Axis.stsState = E_AxisState.Ready AND Z_Axis.stsState = E_AxisState.Ready THEN
			stsCurrentStep := 5020;
		END_IF
	5020: //Home z axis
		Z_Axis.inpPosition := inpZ_HomePos;
		Z_Axis.cmd := E_AxisCommand.ExecuteMoveAbs;
		IF Z_Axis.stsPosition = inpZ_HomePos THEN
			stsCurrentStep := 5030;
		END_IF
	5030: //Home x-axis
		X_Axis.inpPosition := inpX_HomePos;
		X_Axis.cmd := E_AxisCommand.ExecuteMoveAbs;
		IF X_Axis.stsPosition = inpX_HomePos THEN
			stsCurrentStep := 0;
		END_IF
END_CASE
END_METHOD

METHOD Map : BOOL
VAR_INPUT
END_VAR
X_Axis(Axis := AxisX, inpVelocity := 500.0, inpAcceleration := 100.0, inpDeceleration := 100.0);
Z_Axis(Axis := AxisZ, inpVelocity := 500.0, inpAcceleration := 100.0, inpDeceleration := 100.0);
Magnet();
Gripper();

//Handshakes with part conveyor and pallet conveyor
PartConvReady := ipPart.PartReady;
PalletConvReady := ipPallet.PalletReady;
END_METHOD

{warning 'add property implementation'}
PROPERTY PalletReady : BOOL
GET
PalletReady := X_Axis.stsPosition <= inpX_PrePlacePos;
END_GET
END_PROPERTY

{warning 'add property implementation'}
PROPERTY PartPicked : BOOL
GET
PartPicked := Gripper.stsState = E_ActuatorState.AtWork AND Magnet.stsState = E_ActuatorState.AtWork;
END_GET
END_PROPERTY

{warning 'add property implementation'}
PROPERTY PartReady : BOOL
GET
PartReady := Z_Axis.stsPosition <= inpZ_PrePickPos OR X_Axis.stsPosition >= inpX_PrePlacePos;
END_GET
END_PROPERTY

METHOD Picking : BOOL
VAR_INPUT
END_VAR
CASE stsCurrentStep OF
	3000: //Home z-axis
		Z_Axis.inpPosition := inpZ_HomePos;
		Z_Axis.cmd := E_AxisCommand.ExecuteMoveAbs;
		IF Z_Axis.stsPosition = inpZ_HomePos THEN
			stsCurrentStep := 3010;
		END_IF
	3010: //X-axis to pick position
		X_Axis.inpPosition := inpX_PickPos;
		X_Axis.cmd := E_AxisCommand.ExecuteMoveAbs;
		IF X_Axis.stsPosition = inpX_PickPos THEN
			stsCurrentStep := 3020;
		END_IF
	3020: //Z-axis to pre-pick position
		Z_Axis.inpPosition := inpZ_PrePickPos;
		Z_Axis.cmd := E_AxisCommand.ExecuteMoveAbs;
		IF Z_Axis.stsPosition = inpZ_PrePickPos THEN
			stsCurrentStep := 3030;
		END_IF
	3030: //Wait for the conveyor to be ready for pick
		IF PartConvReady THEN
			stsCurrentStep := 3040;
		END_IF
	3040: //Z-axis to pick position
		Z_Axis.inpPosition := inpZ_PickPos;
		Z_Axis.cmd := E_AxisCommand.ExecuteMoveAbs;
		IF Z_Axis.stsPosition = inpZ_PickPos THEN
			stsCurrentStep := 3050;
		END_IF
	3050: //Engage magnets and close grippers
		Magnet.cmd := E_ActuatorCommand.Work;
		Gripper.cmd := E_ActuatorCommand.Work;
		IF Magnet.stsState = E_ActuatorState.AtWork AND Gripper.stsState = E_ActuatorState.AtWork THEN
			stsCurrentStep := 3060;
		END_IF
	3060: //Z-axis to home position
		Z_Axis.inpPosition := inpZ_HomePos;
		Z_Axis.cmd := E_AxisCommand.ExecuteMoveAbs;
		IF Z_Axis.stsPosition = inpZ_HomePos THEN
			stsCurrentStep := 3070;
		END_IF
	3070: //X-axis to pre-place position
		X_Axis.inpPosition := inpX_PrePlacePos;
		X_Axis.cmd := E_AxisCommand.ExecuteMoveAbs;
		IF X_Axis.stsPosition = inpX_PrePlacePos THEN
			stsCurrentStep := 0;
		END_IF
END_CASE
END_METHOD

METHOD Placing : BOOL
VAR_INPUT
END_VAR
VAR
	X_PlacePos				: LREAL;
END_VAR
IF NextPlaceIndex = 1 THEN
	X_PlacePos := inpX_PlacePos1;
ELSIF NextPlaceIndex = 2 THEN
	X_PlacePos := inpX_PlacePos2;
ELSIF NextPlaceIndex = 3 THEN
	X_PlacePos := inpX_PlacePos3;
ELSE
	X_PlacePos := 0;	
END_IF

CASE stsCurrentStep OF
	4000: //Z-axis to home position
		Z_Axis.inpPosition := inpZ_HomePos;
		Z_Axis.cmd := E_AxisCommand.ExecuteMoveAbs;
		IF Z_Axis.stsPosition = inpZ_HomePos THEN
			stsCurrentStep := 4010;
		END_IF
	4010: //X-axis to pre-place position
		X_Axis.inpPosition := inpX_PrePlacePos;
		X_Axis.cmd := E_AxisCommand.ExecuteMoveAbs;
		IF X_Axis.stsPosition = inpX_PrePlacePos THEN
			stsCurrentStep := 4020;
		END_IF
	4020: //Wait for pallet conveyor to be ready for place
		IF PalletConvReady THEN
			stsCurrentStep := 4030;
		END_IF
	4030: //X-axis to place position
		X_Axis.inpPosition := X_PlacePos;
		X_Axis.cmd := E_AxisCommand.ExecuteMoveAbs;
		IF X_Axis.stsPosition = X_PlacePos THEN
			stsCurrentStep := 4035;
		END_IF
	4035: //Z-axis to place position
		Z_Axis.inpPosition := inpZ_PlacePos;
		Z_Axis.cmd := E_AxisCommand.ExecuteMoveAbs;
		IF Z_Axis.stsPosition = inpZ_PlacePos THEN
			stsCurrentStep := 4040;
		END_IF
	4040: //Disengage magnets and grippers
		Magnet.cmd := E_ActuatorCommand.Home;
		Gripper.cmd := E_ActuatorCommand.Home;
		IF Magnet.stsState = E_ActuatorState.AtHome AND Gripper.stsState = E_ActuatorState.AtHome THEN
			stsCurrentStep := 4050;
		END_IF
	4050: //Update data records corresponding to place locations
		IF NextPlaceIndex = 1 THEN
			DataIndex1 := inpDataIndex1;
			DataIndex2 := inpDataIndex2;
		ELSIF NextPlaceIndex = 2 THEN
			DataIndex1 := inpDataIndex3;
			DataIndex2 := inpDataIndex4;
		ELSIF NextPlaceIndex = 3 THEN
			DataIndex1 := inpDataIndex5;
			DataIndex2 := inpDataIndex6;
		END_IF
		IF inpActiveRecord > 0 AND NextPlaceIndex > 0 THEN
			inpPalletRecord[inpActiveRecord].Data[DataIndex1] := 'Part Loaded';
			inpPalletRecord[inpActiveRecord].Data[DataIndex2] := 'Part Loaded';
			stsCurrentStep := 4060;
		END_IF
	4060: //Z-axis to home position
		Z_Axis.inpPosition := inpZ_HomePos;
		Z_Axis.cmd := E_AxisCommand.ExecuteMoveAbs;
		IF Z_Axis.stsPosition = inpZ_HomePos THEN
			stsCurrentStep := 4070;
		END_IF
	4070: //Z-axis to pick position
		X_Axis.inpPosition := inpX_PickPos;
		X_Axis.cmd := E_AxisCommand.ExecuteMoveAbs;
		IF X_Axis.stsPosition = inpX_PickPos THEN
			stsCurrentStep := 0;
		END_IF
END_CASE
END_METHOD

METHOD StateMachine : BOOL
VAR_INPUT
END_VAR
CASE stsState OF
	E_GantryState.Idle: //Module is idle waiting for command
		IF cmd = E_GantryCommand.TurnOn THEN
			stsState := E_GantryState.TurningOn;
		ELSIF cmd = E_GantryCommand.Home THEN
			stsState := E_GantryState.Homing;
		END_IF
	E_GantryState.TurningOn: //Turn on x and z servos
		TurningOn();
		IF stsCurrentStep = 0 AND X_Axis.stsState = E_AxisState.Ready AND Z_Axis.stsState = E_AxisState.Ready THEN
			stsState := E_GantryState.Ready;
		END_IF
	E_GantryState.TurningOff: //Turn off x and z servos
		TurningOff();
		IF stsCurrentStep = 0 AND X_Axis.stsState = E_AxisState.Off AND Z_Axis.stsState = E_AxisState.Off THEN
			stsState := E_GantryState.Idle;
		END_IF
	E_GantryState.Ready: //Gantry ready for command
		IF cmd = E_GantryCommand.Pick THEN
			stsState := E_GantryState.Picking;
		ELSIF cmd = E_GantryCommand.Place THEN
			stsState := E_GantryState.Placing;
		END_IF
	E_GantryState.Homing: //Return gantry to home position
		Homing();
		IF (stsCurrentStep = 0 AND
			X_Axis.stsPosition = inpX_HomePos AND
			Z_Axis.stsPosition = inpZ_HomePos AND
			Gripper.stsState = E_ActuatorState.AtHome AND
			Magnet.stsState = E_ActuatorState.AtHome) 
		THEN
			stsState := E_GantryState.Ready;
		END_IF
	E_GantryState.Picking: //Run pick routine
		Picking();
		IF (stsCurrentStep = 0 AND
			X_Axis.stsPosition = inpX_PrePlacePos AND
			Z_Axis.stsPosition = inpZ_HomePos AND
			Gripper.stsState = E_ActuatorState.AtWork AND
			Magnet.stsState = E_ActuatorState.AtWork) 
		THEN
			stsState := E_GantryState.Placing;
		END_IF
	E_GantryState.Placing: //Run place routine
		Placing();
		IF (stsCurrentStep = 0 AND
			X_Axis.stsPosition = inpX_PickPos AND
			Z_Axis.stsPosition = inpZ_HomePos AND
			Gripper.stsState = E_ActuatorState.AtHome AND
			Magnet.stsState = E_ActuatorState.AtHome) 
		THEN
			stsState := E_GantryState.Ready;
		END_IF
	E_GantryState.Aborting: //Abort current process
		Aborting();
		IF stsCurrentStep = 0 AND X_Axis.stsState <> E_AxisState.Moving AND X_Axis.stsState <> E_AxisState.Moving THEN
			stsState := E_GantryState.Idle;
		END_IF		
END_CASE

IF cmd = E_GantryCommand.Abort THEN
	stsState := E_GantryState.Aborting;
END_IF

cmd := E_GantryCommand.None;
END_METHOD

METHOD Status : BOOL
VAR_INPUT
END_VAR
//Determine next place location depending on current data records
IF inpPalletRecord[inpActiveRecord].Data[inpDataIndex1] = '' AND inpPalletRecord[inpActiveRecord].Data[inpDataIndex2] = '' THEN
	NextPlaceIndex := 1;
ELSIF inpPalletRecord[inpActiveRecord].Data[inpDataIndex3] = '' AND inpPalletRecord[inpActiveRecord].Data[inpDataIndex4] = '' THEN
	NextPlaceIndex := 2;
ELSIF inpPalletRecord[inpActiveRecord].Data[inpDataIndex5] = '' AND inpPalletRecord[inpActiveRecord].Data[inpDataIndex6] = '' THEN
	NextPlaceIndex := 3;
ELSE
	NextPlaceIndex := 0;
END_IF

//If ready, auto command pick sequence
IF inpActiveRecord <> 0 AND NextPlaceIndex > 0 AND stsState = E_GantryState.Ready THEN
	stsState := E_GantryState.Picking;
END_IF

//State transition one shots
rtTurningOn(CLK := stsState = E_GantryState.TurningOn);
IF rtTurningOn.Q THEN
	stsCurrentStep := 1000;
END_IF

rtTurningOff(CLK := stsState = E_GantryState.TurningOff);
IF rtTurningOff.Q THEN
	stsCurrentStep := 2000;
END_IF

rtPicking(CLK := stsState = E_GantryState.Picking);
IF rtPicking.Q THEN
	stsCurrentStep := 3000;
END_IF

rtPlacing(CLK := stsState = E_GantryState.Placing);
IF rtPlacing.Q THEN
	stsCurrentStep := 4000;
END_IF

rtHoming(CLK := stsState = E_GantryState.Homing);
IF rtHoming.Q THEN
	stsCurrentStep := 5000;
END_IF
END_METHOD

METHOD TurningOff : BOOL
VAR_INPUT
END_VAR
CASE stsCurrentStep OF
	2000: //Turn off x and z axes
		X_Axis.cmd := E_AxisCommand.TurnOff;
		Z_Axis.cmd := E_AxisCommand.TurnOff;
		IF X_Axis.stsState = E_AxisState.Off AND Z_Axis.stsState = E_AxisState.Off THEN
			stsCurrentStep := 0;
		END_IF
END_CASE
END_METHOD

METHOD TurningOn : BOOL
VAR_INPUT
END_VAR
CASE stsCurrentStep OF
	1000: //Turn on x and z axes
		X_Axis.cmd := E_AxisCommand.TurnOn;
		Z_Axis.cmd := E_AxisCommand.TurnOn;
		IF X_Axis.stsState = E_AxisState.Ready AND Z_Axis.stsState = E_AxisState.Ready THEN
			stsCurrentStep := 0;
		END_IF
END_CASE
END_METHOD

END_FUNCTION_BLOCK
